// TIA Portal project "EMA3135 51_SCC" (V16)

(* hardware
DEVICE "PC-System_1"  SIMATIC PC station
   slot 0: "SIMATIC PC station"  Rail  SIMATIC PC-Station  V1.0
      slot 125: "Stationmanager"  Station_Manager  V6.0.4
   slot 1: "HMI_RT_1"  WinCC RT Professional  6AV2 105-0xxxx-xxxx  16.0.0.0
   slot 2: "IE general_1"  IE General  IE_CP  V8.2.0
DEVICE "S7-1200 station_1"  S7-1200 Station
   slot 0: "Rack_0"  S7-1200 Rack  Rack  V1.0
   slot 1: "PLC_1"  CPU 1214C AC/DC/Rly  6ES7 214-1BG40-0XB0  V4.2
*)

// ===== PLC "PLC_1"  CPU 1214C AC/DC/Rly =====

VAR_GLOBAL   // PLC tag table "Default tag table"
   "START" AT %I0.0 : Bool;
   "STOP" AT %I0.1 : Bool;
   "MODE" AT %I0.2 : Bool;
   "SENSOR_1" AT %I0.3 : Bool;
   "SENSOR_2" AT %I0.4 : Bool;
   "SENSOR_3" AT %I0.5 : Bool;
   "SENSOR_4" AT %I0.6 : Bool;
   "SENSOR_5" AT %I0.7 : Bool;
   "SENSOR_6" AT %I1.0 : Bool;
   "SENSOR_7" AT %I1.1 : Bool;
   "SENSOR_8" AT %I1.2 : Bool;
   "CONVEYOR_BELT_1" AT %Q0.0 : Bool;
   "CONVEYOR_BELT_2" AT %Q0.1 : Bool;
   "CONVEYOR_BELT_3" AT %Q0.2 : Bool;
   "CONVEYOR_BELT_4_L" AT %Q0.3 : Bool;
   "CONVEYOR_BELT_4_R" AT %Q0.4 : Bool;
   "CONTAINER_1_FULL" AT %Q0.5 : Bool;
   "CONTAINER_2_FULL" AT %Q0.6 : Bool;
   "MODE_1" AT %M1.3 : Bool;
   "MODE_2" AT %M2.0 : Bool;
   "Memory 2" AT %M1.5 : Bool;
   "Memory 1" AT %M1.6 : Bool;
   "Memory 3" AT %M1.7 : Bool;
   "Sim" AT %I1.3 : Bool;
   "Box1_1" AT %MD0 : DWord;
   "Box3_1" AT %MD2 : DWord;
   "Box2_1" AT %MD1 : DWord;
   "Box1_2" AT %MD3 : DWord;
   "Box2_2" AT %MD4 : DWord;
   "Box3_2" AT %MD5 : DWord;
   "sim_senor1" AT %M9.0 : Bool;
   "sim_senor2" AT %M9.1 : Bool;
END_VAR

// folder: System blocks/Program resources

DATA_BLOCK "IEC_Counter_0_DB"   // DB1
{ S7_Optimized_Access := 'TRUE' }
AUTHOR : Simatic
FAMILY : IEC
NAME : CNTR
VERSION : 1.0
// stored: InstanceOfName IEC_COUNTER
"IEC_COUNTER"
BEGIN
END_DATA_BLOCK

DATA_BLOCK "IEC_Counter_0_DB_1"   // DB2
{ S7_Optimized_Access := 'TRUE' }
AUTHOR : Simatic
FAMILY : IEC
NAME : CNTR
VERSION : 1.0
// stored: InstanceOfName IEC_COUNTER
"IEC_COUNTER"
BEGIN
END_DATA_BLOCK

DATA_BLOCK "IEC_Counter_0_DB_2"   // DB3
{ S7_Optimized_Access := 'TRUE' }
AUTHOR : Simatic
FAMILY : IEC
NAME : CNTR
VERSION : 1.0
// stored: InstanceOfName IEC_COUNTER
"IEC_COUNTER"
BEGIN
END_DATA_BLOCK

DATA_BLOCK "IEC_Counter_0_DB_3"   // DB4
{ S7_Optimized_Access := 'TRUE' }
AUTHOR : Simatic
FAMILY : IEC
NAME : CNTR
VERSION : 1.0
// stored: InstanceOfName IEC_COUNTER
"IEC_COUNTER"
BEGIN
END_DATA_BLOCK

DATA_BLOCK "IEC_Counter_0_DB_4"   // DB5
{ S7_Optimized_Access := 'TRUE' }
AUTHOR : Simatic
FAMILY : IEC
NAME : CNTR
VERSION : 1.0
// stored: InstanceOfName IEC_COUNTER
"IEC_COUNTER"
BEGIN
END_DATA_BLOCK

DATA_BLOCK "IEC_Counter_0_DB_5"   // DB6
{ S7_Optimized_Access := 'TRUE' }
AUTHOR : Simatic
FAMILY : IEC
NAME : CNTR
VERSION : 1.0
// stored: InstanceOfName IEC_COUNTER
"IEC_COUNTER"
BEGIN
END_DATA_BLOCK

DATA_BLOCK "IEC_Timer_0_DB"   // DB7
{ S7_Optimized_Access := 'TRUE' }
AUTHOR : Simatic
FAMILY : IEC
NAME : IEC_TMR
VERSION : 1.0
// stored: InstanceOfName IEC_TIMER
"IEC_TIMER"
BEGIN
END_DATA_BLOCK

DATA_BLOCK "IEC_Timer_0_DB_1"   // DB8
{ S7_Optimized_Access := 'TRUE' }
AUTHOR : Simatic
FAMILY : IEC
NAME : IEC_TMR
VERSION : 1.0
// stored: InstanceOfName IEC_TIMER
"IEC_TIMER"
BEGIN
END_DATA_BLOCK

// folder: (top level)

ORGANIZATION_BLOCK "Main"   // OB1, LAD, ProgramCycle
TITLE = "Main Program Sweep (Cycle)"
{ S7_Optimized_Access := 'TRUE' }
VERSION : 0.1
   VAR_INPUT
      Initial_Call : Bool;   // Initial call of this OB
      Remanence : Bool;   // =True, if remanent data are available
   END_VAR
   VAR_TEMP
      resetcounter3 : Bool;
      resetcounter5 : Bool;
      resetcounter2 : Bool;
      resetcounter4 : Bool;
      Box3_1 : Time;
      Box1_1 : Time;
      Box2_1 : Time;
   END_VAR
   VAR_TEMP   // added for the SCL form of the ladder/FBD networks
      _w1 : Bool;
      _w2 : Bool;
   END_VAR
BEGIN

REGION Network 1: Choose mode and reset container and counter
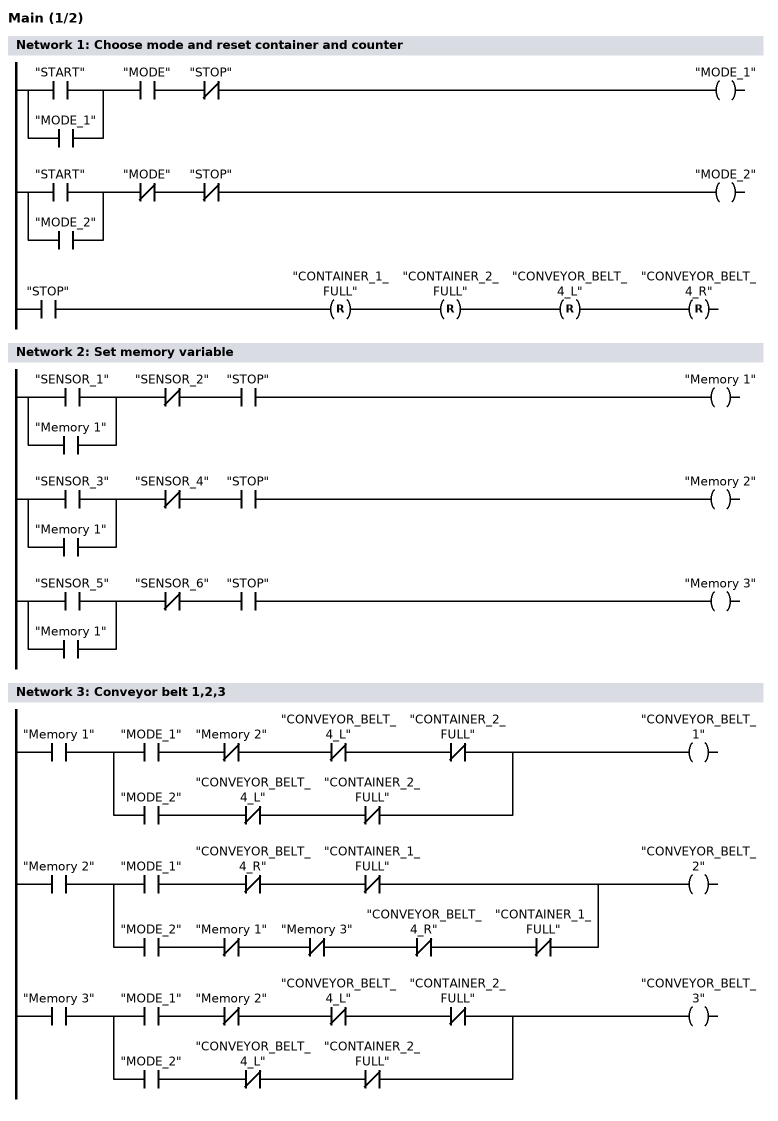
   RUNG wire#powerrail
      Contact( "START" )
      wire#w1
      Contact( "MODE" )
      I_Contact( "STOP" )
      Coil( "MODE_1" )
   END_RUNG
   RUNG wire#powerrail
      Contact( "MODE_1" )
   END_RUNG wire#w1
   RUNG wire#powerrail
      Contact( "START" )
      wire#w2
      I_Contact( "MODE" )
      I_Contact( "STOP" )
      Coil( "MODE_2" )
   END_RUNG
   RUNG wire#powerrail
      Contact( "MODE_2" )
   END_RUNG wire#w2
   RUNG wire#powerrail
      Contact( "STOP" )
      R_Coil( "CONTAINER_1_FULL" )
      R_Coil( "CONTAINER_2_FULL" )
      R_Coil( "CONVEYOR_BELT_4_L" )
      R_Coil( "CONVEYOR_BELT_4_R" )
   END_RUNG
   // the same network as SCL:
   "MODE_1" := ("START" OR "MODE_1") AND "MODE" AND NOT "STOP";
   "MODE_2" := ("START" OR "MODE_2") AND NOT "MODE" AND NOT "STOP";
   IF "STOP" THEN
       "CONTAINER_1_FULL" := FALSE;
       "CONTAINER_2_FULL" := FALSE;
       "CONVEYOR_BELT_4_L" := FALSE;
       "CONVEYOR_BELT_4_R" := FALSE;
   END_IF;
END_REGION

REGION Network 2: Set memory variable
   RUNG wire#powerrail
      Contact( "SENSOR_1" )
      wire#w1
      I_Contact( "SENSOR_2" )
      Contact( "STOP" )
      Coil( "Memory 1" )
   END_RUNG
   RUNG wire#powerrail
      Contact( "Memory 1" )
   END_RUNG wire#w1
   RUNG wire#powerrail
      Contact( "SENSOR_3" )
      wire#w2
      I_Contact( "SENSOR_4" )
      Contact( "STOP" )
      Coil( "Memory 2" )
   END_RUNG
   RUNG wire#powerrail
      Contact( "Memory 1" )
   END_RUNG wire#w2
   RUNG wire#powerrail
      Contact( "SENSOR_5" )
      wire#w3
      I_Contact( "SENSOR_6" )
      Contact( "STOP" )
      Coil( "Memory 3" )
   END_RUNG
   RUNG wire#powerrail
      Contact( "Memory 1" )
   END_RUNG wire#w3
   // the same network as SCL:
   "Memory 1" := ("SENSOR_1" OR "Memory 1") AND NOT "SENSOR_2" AND "STOP";
   "Memory 2" := ("SENSOR_3" OR "Memory 1") AND NOT "SENSOR_4" AND "STOP";
   "Memory 3" := ("SENSOR_5" OR "Memory 1") AND NOT "SENSOR_6" AND "STOP";
END_REGION

REGION Network 3: Conveyor belt 1,2,3
   RUNG wire#powerrail
      Contact( "Memory 1" )
      wire#w1
      Contact( "MODE_1" )
      I_Contact( "Memory 2" )
      I_Contact( "CONVEYOR_BELT_4_L" )
      I_Contact( "CONTAINER_2_FULL" )
      wire#w2
      Coil( "CONVEYOR_BELT_1" )
   END_RUNG
   RUNG wire#w1
      Contact( "MODE_2" )
      I_Contact( "CONVEYOR_BELT_4_L" )
      I_Contact( "CONTAINER_2_FULL" )
   END_RUNG wire#w2
   RUNG wire#powerrail
      Contact( "Memory 2" )
      wire#w3
      Contact( "MODE_1" )
      I_Contact( "CONVEYOR_BELT_4_R" )
      I_Contact( "CONTAINER_1_FULL" )
      wire#w4
      Coil( "CONVEYOR_BELT_2" )
   END_RUNG
   RUNG wire#w3
      Contact( "MODE_2" )
      I_Contact( "Memory 1" )
      I_Contact( "Memory 3" )
      I_Contact( "CONVEYOR_BELT_4_R" )
      I_Contact( "CONTAINER_1_FULL" )
   END_RUNG wire#w4
   RUNG wire#powerrail
      Contact( "Memory 3" )
      wire#w5
      Contact( "MODE_1" )
      I_Contact( "Memory 2" )
      I_Contact( "CONVEYOR_BELT_4_L" )
      I_Contact( "CONTAINER_2_FULL" )
      wire#w6
      Coil( "CONVEYOR_BELT_3" )
   END_RUNG
   RUNG wire#w5
      Contact( "MODE_2" )
      I_Contact( "CONVEYOR_BELT_4_L" )
      I_Contact( "CONTAINER_2_FULL" )
   END_RUNG wire#w6
   // the same network as SCL:
   "CONVEYOR_BELT_1" := "Memory 1" AND (("MODE_1" AND NOT "Memory 2" AND NOT "CONVEYOR_BELT_4_L" AND NOT "CONTAINER_2_FULL") OR ("MODE_2" AND NOT "CONVEYOR_BELT_4_L" AND NOT "CONTAINER_2_FULL"));
   "CONVEYOR_BELT_2" := "Memory 2" AND (("MODE_1" AND NOT "CONVEYOR_BELT_4_R" AND NOT "CONTAINER_1_FULL") OR ("MODE_2" AND NOT "Memory 1" AND NOT "Memory 3" AND NOT "CONVEYOR_BELT_4_R" AND NOT "CONTAINER_1_FULL"));
   "CONVEYOR_BELT_3" := "Memory 3" AND (("MODE_1" AND NOT "Memory 2" AND NOT "CONVEYOR_BELT_4_L" AND NOT "CONTAINER_2_FULL") OR ("MODE_2" AND NOT "CONVEYOR_BELT_4_L" AND NOT "CONTAINER_2_FULL"));
END_REGION

REGION Network 4: Conveyor belt 4
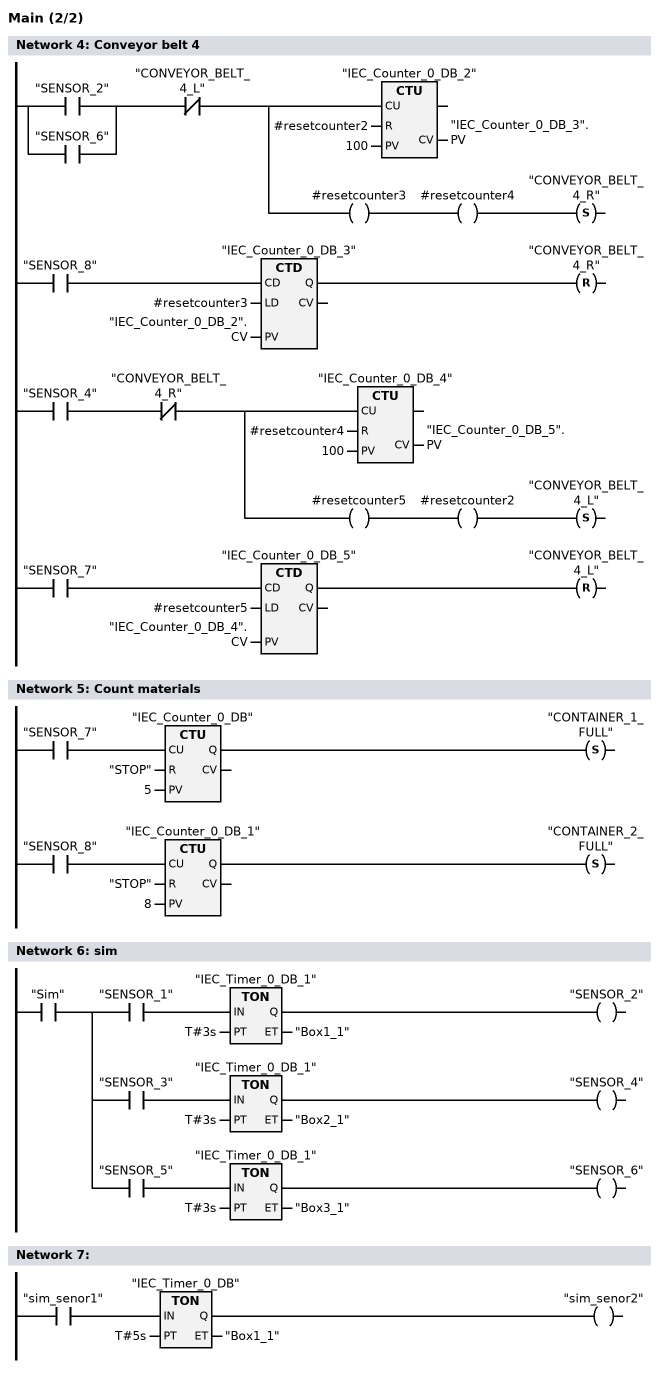
   #_w1 := ("SENSOR_2" OR "SENSOR_6") AND NOT "CONVEYOR_BELT_4_L";
   "IEC_Counter_0_DB_2".CTU(CU := #_w1, R := #resetcounter2, PV := 100, CV => "IEC_Counter_0_DB_3".PV);
   #resetcounter3 := #_w1;
   #resetcounter4 := #_w1;
   IF #_w1 THEN "CONVEYOR_BELT_4_R" := TRUE; END_IF;
   "IEC_Counter_0_DB_3".CTD(CD := "SENSOR_8", LD := #resetcounter3, PV := "IEC_Counter_0_DB_2".CV);
   IF "IEC_Counter_0_DB_3".Q THEN "CONVEYOR_BELT_4_R" := FALSE; END_IF;
   #_w2 := "SENSOR_4" AND NOT "CONVEYOR_BELT_4_R";
   "IEC_Counter_0_DB_4".CTU(CU := #_w2, R := #resetcounter4, PV := 100, CV => "IEC_Counter_0_DB_5".PV);
   #resetcounter5 := #_w2;
   #resetcounter2 := #_w2;
   IF #_w2 THEN "CONVEYOR_BELT_4_L" := TRUE; END_IF;
   "IEC_Counter_0_DB_5".CTD(CD := "SENSOR_7", LD := #resetcounter5, PV := "IEC_Counter_0_DB_4".CV);
   IF "IEC_Counter_0_DB_5".Q THEN "CONVEYOR_BELT_4_L" := FALSE; END_IF;
END_REGION

REGION Network 5: Count materials
   "IEC_Counter_0_DB".CTU(CU := "SENSOR_7", R := "STOP", PV := 5);
   IF "IEC_Counter_0_DB".Q THEN "CONTAINER_1_FULL" := TRUE; END_IF;
   "IEC_Counter_0_DB_1".CTU(CU := "SENSOR_8", R := "STOP", PV := 8);
   IF "IEC_Counter_0_DB_1".Q THEN "CONTAINER_2_FULL" := TRUE; END_IF;
END_REGION

REGION Network 6: sim
   "IEC_Timer_0_DB_1".TON(IN := "Sim" AND "SENSOR_1", PT := T#3s, ET => "Box1_1");
   "SENSOR_2" := "IEC_Timer_0_DB_1".Q;
   "IEC_Timer_0_DB_1".TON(IN := "Sim" AND "SENSOR_3", PT := T#3s, ET => "Box2_1");
   "SENSOR_4" := "IEC_Timer_0_DB_1".Q;
   "IEC_Timer_0_DB_1".TON(IN := "Sim" AND "SENSOR_5", PT := T#3s, ET => "Box3_1");
   "SENSOR_6" := "IEC_Timer_0_DB_1".Q;
END_REGION

REGION Network 7
   "IEC_Timer_0_DB".TON(IN := "sim_senor1", PT := T#5s, ET => "Box1_1");
   "sim_senor2" := "IEC_Timer_0_DB".Q;
END_REGION
END_ORGANIZATION_BLOCK

(* ===== HMI "HMI_RT_1" =====
system functions are stored by id; their names below are inferred from use
connection "HMI_Connection_1": S71200_TCP_IP, SCADA_S7_1200

HMI tags "Default tag table"
   "START" : Bool = PLC START AT %I0.0, 500 ms
   "SENSOR_3" : Bool = PLC SENSOR_3 AT %I0.5, 500 ms
   "MODE" : Bool = PLC MODE AT %I0.2, 500 ms
   "STOP" : Bool = PLC STOP AT %I0.1, 500 ms
   "CONVEYOR_BELT_2" : Bool = PLC CONVEYOR_BELT_2 AT %Q0.1, 500 ms
   "MODE_1" : Bool = PLC MODE_1 AT %M1.3, 500 ms
   "Memory2" : Bool = PLC "Memory 2" AT %M1.5, 500 ms
   "Memory1" : Bool = PLC "Memory 1" AT %M1.6, 500 ms
   "Memory3" : Bool = PLC "Memory 3" AT %M1.7, 500 ms
   "Box3_1" : DWord = PLC Box3_1 AT %MD2, 500 ms
   "SENSOR_5" : Bool = PLC SENSOR_5 AT %I0.7, 500 ms
   "SENSOR_6" : Bool = PLC SENSOR_6 AT %I1.0, 500 ms
   "SENSOR_2" : Bool = PLC SENSOR_2 AT %I0.4, 500 ms
   "MODE_2" : Bool = PLC MODE_2 AT %M2.0, 500 ms
   "Sim" : Bool = PLC Sim AT %I1.3, 500 ms
   "sim_senor1" : Bool = PLC sim_senor1 AT %M9.0, 500 ms
   "Box1_1" : DWord = PLC Box1_1 AT %MD0, 500 ms

screen "Home" 1024x768
   GraphicView "Graphic view_2" at 327,323 size 676x303; Picture "Graphic_7"
   Clock "Clock_1" at 0,0 size 128x128
   DiskSpaceView "Memory space view_1" at 153,28 size 60x100
   TextField "Text field_1" at 133,5 size 91x19; Text 'Memory space'
   Button "Button_1" at 877,39 size 108x50; TextOff 'Exit'
      on Click: StopRuntime(0)
   TextField "Text field_2" at 241,20 size 279x78; Text 'Ho va Ten: Pham Quang Vinh MSSV: 21021392 Module: N-PLCE-SCC'
   TextField "Text field_3" at 48,141 size 95x19; Text 'Control Panel'
   GraphicView "Graphic view_1" at 428,329 size 421x73; Picture "Graphic_6"
   GraphicView "Graphic view_5" at 230,427 size 421x73; Picture "Graphic_6"
      Appearance <- "Memory2"
   GraphicView "Graphic view_6" at 6,539 size 421x73; Picture "Graphic_6"
      Appearance <- "Memory3"
   GraphicView "Graphic view_4" at 897,356 size 127x73; Picture "Graphic_12"
   GraphicView "Graphic view_3" at 464,289 size 127x77; Picture "Graphic_8"
      HorizontalMovement <- "Box1_1"
   GraphicView "Graphic view_7" at 353,616 size 127x73; Picture "Graphic_12"
   GraphicView "Graphic view_12" at 267,386 size 127x77; Picture "Graphic_8"
      Appearance <- "SENSOR_3"
   GraphicView "Graphic view_13" at 39,500 size 127x77; Picture "Graphic_8"
      HorizontalMovement <- "Box3_1"
   SymbolLibrary "Symbol library_1" at 523,231 size 27x54
   SymbolLibrary "Symbol library_2" at 786,231 size 27x54
      Appearance <- "SENSOR_2"
   SymbolLibrary "Symbol library_3" at 326,327 size 27x54
      Appearance <- "SENSOR_3"
   SymbolLibrary "Symbol library_4" at 589,327 size 27x54
   SymbolLibrary "Symbol library_5" at 92,445 size 27x54
      Appearance <- "SENSOR_5"
   SymbolLibrary "Symbol library_6" at 355,445 size 27x54
      Appearance <- "SENSOR_6"
   TextField "Text field_4" at 436,392 size 92x22; Text 'Conveyor 1'
   TextField "Text field_5" at 240,490 size 93x22; Text 'Conveyor 2'
   TextField "Text field_6" at 15,601 size 97x22; Text 'Conveyor 3'
   TextField "Text field_7" at 765,500 size 92x22; Text 'Conveyor 4'
   TextField "Text field_8" at 509,206 size 62x19; Text 'Sensor 1'
   TextField "Text field_9" at 769,207 size 62x19; Text 'Sensor 2'
   TextField "Text field_10" at 310,305 size 62x19; Text 'Sensor 3'
   TextField "Text field_11" at 570,306 size 62x19; Text 'Sensor 4'
   TextField "Text field_12" at 77,421 size 62x19; Text 'Sensor 5'
   TextField "Text field_13" at 337,422 size 62x19; Text 'Sensor 6'
   SymbolLibrary "Symbol library_7" at 965,309 size 54x27
   SymbolLibrary "Symbol library_8" at 509,591 size 54x32
   GraphicView "Graphic view_8" at 825,283 size 127x77; Picture "Graphic_8"
   TextField "Text field_14" at 581,601 size 62x19; Text 'Sensor 7'
   TextField "Text field_15" at 959,285 size 62x19; Text 'Sensor 8'
   Button "Button_2" at 302,276 size 80x30; TextOff 'Sensor 3'
      on PressLeft: SetBit("SENSOR_3")
      on ReleaseLeft: ResetBit("SENSOR_3")
   Button "Button_3" at 15,175 size 50x40; TextOff 'Start'
      on PressLeft: SetBit("START")
      on ReleaseLeft: ResetBit("START")
   Button "Button_4" at 75,175 size 50x40; TextOff 'Stop'
      on PressLeft: SetBit("STOP")
      on ReleaseLeft: ResetBit("STOP")
   Button "Button_5" at 136,175 size 50x40; TextOff 'Mode'
      on PressLeft: SetBit("MODE")
      on ReleaseLeft: ResetBit("MODE")
      Appearance <- "MODE"
   Button "Button_6" at 68,391 size 80x30; TextOff 'Sensor 5'
      on PressLeft: SetBit("SENSOR_3")
      on ReleaseLeft: ResetBit("SENSOR_3")
   Button "Button_7" at 495,175 size 80x30; TextOff 'Sensor 1'
      on PressLeft: SetBit("sim_senor1")
      on ReleaseLeft: ResetBit("sim_senor1")
   Button "Button_8" at 213,175 size 50x40; TextOff 'Sim'
      on PressLeft: SetBit("Sim")
      on ReleaseLeft: ResetBit("Sim")
   RoundButton "Round button_1" at 278,167 size 48x48; Text 'Text'
      Appearance <- "MODE_1"
   RoundButton "Round button_2" at 341,167 size 48x48; Text 'Text'
      Appearance <- "MODE_2"
   TextField "Text field_16" at 206,151 size 72x19; Text 'Sim mode'
   TextField "Text field_17" at 294,179 size 10x19; Text '1'
   TextField "Text field_18" at 359,180 size 10x19; Text '2'
*)